// TIA Portal V20 export
TYPE "typeDataToSafety"
// Information sent from the standard program to the safety program
// stored: Access Published, IsFailsafeCompliant true, Namespace Safety
   STRUCT
      ackSafetyFromHmi : Int;   // Acknowledge variable from operator control or monitoring system
      ackSafetyGlobal : Bool;   // Acknowledge command to ack all safety
      ackFromUnit1 : Bool;   // Acknowledge command coming from Unit 1
      ackSafetyFromMobileHMI : Bool;   // Acknowledge command coming from Mobile Panel
      resetSafetyFromMobileHMI : Bool;   // Reset command coming from Mobile Panel
      connectionBoxID_1 : Int;   // Mobile Panel Connection Box ID (extend list as needed)
      connectionBoxID_2 : Int;   // Mobile Panel Connection Box ID (extend list as needed)
      MobilePanelConnected : Bool;   // TRUE: connection box is connected
      MobilePanelPermissions : Bool;   // Transfer to Phmi Permissions
      DeselectBA10 : Bool;   // BA10 is not selected and no supply part
      DeselectBA15 : Bool;   // BA15 is not selected and no supply part
      DeselectBA30 : Bool;   // BA30 is not selected and no supply part
      DeselectBA60 : Bool;   // BA60 is not selected and no supply part
      PowerOnCommand : Bool;   // Power On Command
      InitializeEnable : Bool;
      BA060STOP : Bool;   // Stop Done For BA060 Request
      SepaGripperAxisXmoveToBa60 : Bool;
      unitMode : "Safety.typeUnitMode";   // Current mode of the unit
      unitState : "Safety.typeUnitStatus";   // Current States of the unit
      winderUsed : "Safety.typeWinderUseMode";
      StackDoor1 { S7_SetPoint := 'True'} : "Safety.typeFdoorCommands";
      StackDoor2 { S7_SetPoint := 'True'} : "Safety.typeFdoorCommands";
      StackDoor3 { S7_SetPoint := 'True'} : "Safety.typeFdoorCommands";
      StackDoor4 { S7_SetPoint := 'True'} : "Safety.typeFdoorCommands";
      StackDoor5 { S7_SetPoint := 'True'} : "Safety.typeFdoorCommands";
      StackDoor6 { S7_SetPoint := 'True'} : "Safety.typeFdoorCommands";
      StackDoor7 { S7_SetPoint := 'True'} : "Safety.typeFdoorCommands";
      StackDoor8 { S7_SetPoint := 'True'} : "Safety.typeFdoorCommands";
      StackDoor9 { S7_SetPoint := 'True'} : "Safety.typeFdoorCommands";
      StackDoor10 { S7_SetPoint := 'True'} : "Safety.typeFdoorCommands";
      StackDoor12 { S7_SetPoint := 'True'} : "Safety.typeFdoorCommands";
      hotWireCutterCmds : "Safety.typeHotWireCutter";
      clock { ExternalAccessible := 'False'; ExternalVisible := 'False'; ExternalWritable := 'False'} : "Safety.typeGlobalClockMem";
      BrakeTest { S7_SetPoint := 'True'} : "Safety.typeBrakeTest";
   END_STRUCT;
   // // StackDoor1.Lock : zone1Fdoor1Lock
   // // StackDoor1.Unlock : zone1Fdoor1Unock
   // // StackDoor2.Lock : zone1Fdoor2Lock
   // // StackDoor2.Unlock : zone1Fdoor2Unock
   // // StackDoor3.Lock : zone1Fdoor2Lock
   // // StackDoor3.Unlock : zone1Fdoor2Unock
   // // StackDoor4.Lock : zone1Fdoor2Lock
   // // StackDoor4.Unlock : zone1Fdoor2Unock
   // // StackDoor5.Lock : zone1Fdoor2Lock
   // // StackDoor5.Unlock : zone1Fdoor2Unock
   // // StackDoor6.Lock : zone1Fdoor2Lock
   // // StackDoor6.Unlock : zone1Fdoor2Unock
   // // StackDoor7.Lock : zone1Fdoor2Lock
   // // StackDoor7.Unlock : zone1Fdoor2Unock
   // // StackDoor8.Lock : zone1Fdoor2Lock
   // // StackDoor8.Unlock : zone1Fdoor2Unock
   // // StackDoor9.Lock : zone1Fdoor2Lock
   // // StackDoor9.Unlock : zone1Fdoor2Unock
   // // StackDoor10.Lock : zone1Fdoor7Lock
   // // StackDoor10.Unlock : zone1Fdoor7Unock
   // // StackDoor12.Lock : zone1Fdoor9Lock
   // // StackDoor12.Unlock : zone1Fdoor9Unock
END_TYPE
